PROGRAM RunGRAB
VAR
END_VAR

END_PROGRAM

(* stored: Version 1.1.0.1, ProductVersion 3.1.4024.6
   POU RunGRAB: Id {73d75011-4d6e-43ad-a6ea-3904f1e24ffa}, SpecialFunc None *)
